FUNCTION_BLOCK SomeMachine IMPLEMENTS ITF_PackMLMachine
VAR
	_Aborting : Aborting := (MyNextState := _Aborted);
	_Aborted : Aborted := (MyNextState := _Clearing);
	_Clearing : Clearing := (MyNextState := _Stopped, AbortingState := _Aborting);
	_Stopping : Stopping := (MyNextState := _Stopped, AbortingState := _Aborting);
	_Stopped : Stopped := (MyNextState := _Resetting, AbortingState := _Aborting);
	_Resetting : Resetting := (MyNextState := _Idle, AbortingState := _Aborting, StoppingState := _Stopping);
	_Idle : Idle := (MyNextState := _Starting, AbortingState := _Aborting, StoppingState := _Stopping);
	_Starting : Starting := (MyNextState := _Execute, AbortingState := _Aborting, StoppingState := _Stopping);
	_Execute : Execute := (AbortingState := _Aborting, StoppingState := _Stopping);
	_MyState : ITF_PackMLState := _Aborting;
	Initialised: BOOL;
	CurrentState : STRING(20);
END_VAR

METHOD ChangeState : BOOL
VAR_INPUT
	NewState : ITF_PackMLState;
END_VAR
_MyState := NewState;
_MyState.SetContext(this^);
END_METHOD

METHOD CyclicLogic : BOOL
VAR_INPUT
END_VAR
IF NOT Initialised THEN
	_MyState.SetContext(THIS^);
	Initialised := TRUE;
ELSE
	RETURN;
END_IF
IF _MyState <> 0 THEN
	_MyState.CyclicLogic();
	CurrentState := _MyState.MyStateName;
END_IF
END_METHOD

METHOD EStop : BOOL
VAR_INPUT
END_VAR
IF _MyState <> 0 THEN
	_MyState.EStop();
END_IF
END_METHOD

METHOD Reset : BOOL
VAR_INPUT
END_VAR
IF _MyState <> 0 THEN
	_MyState.Reset();
END_IF
END_METHOD

METHOD Start : BOOL
VAR_INPUT
END_VAR
IF _MyState <> 0 THEN
	_MyState.Start();
END_IF
END_METHOD

METHOD Stop : BOOL
VAR_INPUT
END_VAR
IF _MyState <> 0 THEN
	_MyState.Stop();
END_IF
END_METHOD

END_FUNCTION_BLOCK

(* stored: Version 1.1.0.1, ProductVersion 3.1.4024.12
   POU SomeMachine: Id {ff6886fb-65b8-468b-be70-46b545e120bf}, SpecialFunc None
   Method ChangeState: Id {6244edf1-c088-4089-92f0-602943a02aa6}
   Method CyclicLogic: Id {cf8cfe0e-a409-463c-bd73-24a121647ac1}
   Method EStop: Id {1b9f0e87-8745-482b-952c-e92621ee9951}
   Method Reset: Id {64845523-7ded-4c82-a4b2-e98329962d21}
   Method Start: Id {a046d53a-bea4-4b2d-8cec-0d466afe4469}
   Method Stop: Id {feb16b1c-88f9-4336-83ab-82109a72bbc3} *)
